// TIA Portal V17 export
// export: Created 2026-04-13T11:12:41.6152652Z, ExportSetting WithDefaults, DisplayName Totally Integrated Automation Portal, DisplayVersion V17 Update 4, DisplayName TIA Portal Openness, DisplayVersion V17 Update 4, DisplayName TIA Portal Version Control Interface, DisplayVersion V17, DisplayName SINAMICS Startdrive Advanced, DisplayVersion V17, DisplayName SINAMICS Startdrive G130, G150, S120, S150, SINAMICS MV, S210, DisplayVersion V17, DisplayName SINAMICS Startdrive G110M, G120, G120C, G120D, G120P, G115D, DisplayVersion V17, DisplayName STEP 7 Professional, DisplayVersion V17 Update 4, DisplayName STEP 7 Safety, DisplayVersion V17, DisplayName WinCC Professional, DisplayVersion V17 Update 4
FUNCTION_BLOCK "A4-蠕动泵控制"   // FB9, SCL
{ S7_Optimized_Access := 'TRUE' }
VERSION : 0.1
// stored: AutoNumber true, IsIECCheckEnabled false, IsRetainMemResEnabled false, MemoryReserve 100, SetENOAutomatically false, UDAEnableTagReadback false
   VAR_INPUT
      HMI上限 : Real := 50.0;
      HMI下限 : Real;
      PLC上限 : Int := 27648;
      PLC下限 : Int := 0;
      泵报警信号 : Bool;
      泵输入电流 : Int;
   END_VAR
   VAR_OUTPUT
      泵输出反馈 : Real;
      泵报警输出 : Bool;
   END_VAR
   VAR_IN_OUT
      模式设定 : Real;
      泵控制按钮 : Bool;
      频率设定 : Real;
      泵输出Q : Bool;
      泵速度AO : Int;
      安全停机 : Bool;
      泵正反转按钮 : Bool;
      泵正反输出 : Bool;
      动画 : Int;
   END_VAR
   VAR
      Temp_1 : Int;
      DBD1 : Real;
      DBD2 : Real;
      DBD3 : Real;
   END_VAR
BEGIN

   //手动控制--------------------------------------------------------------------------------------------------------------
   IF #模式设定 = 2.0 OR #模式设定 = 3.0 OR #模式设定 = 4.0 THEN
       //预热器加热手动控制
       IF #泵控制按钮 THEN
           #泵输出Q := TRUE;
           (* #泵速度AO := REAL_TO_INT((#频率设定 - #工程下限) * (#模拟高限 - #模拟低限) / (#工程上限 - #工程下限) + #模拟低限); *)
           (* #泵速度AO := REAL_TO_INT(#频率设定 * 27648.0 / 50.0); *)
           #DBD1 := NORM_X_REAL(MIN := #HMI下限, VALUE := #频率设定, MAX := #HMI上限);
           #泵速度AO := SCALE_X_INT(MIN := #PLC下限, VALUE := #DBD1, MAX := #PLC上限);
       ELSE
           #泵输出Q := FALSE;
       END_IF;

       IF #泵正反转按钮 THEN
           #泵正反输出 := 1;
       ELSE
           #泵正反输出 := 0;
       END_IF;
   END_IF;

   //自动启动--------------------------------------------------------------------------------------------------------------


   IF #模式设定 = 1.0 THEN
       (* #泵速度AO := REAL_TO_INT((#频率设定 - #工程下限) * (#模拟高限 - #模拟低限) / (#工程上限 - #工程下限) + #模拟低限); *)
       (* #泵速度AO := REAL_TO_INT(#频率设定 * 27648.0 / 50.0); *)
       #DBD2 := NORM_X_REAL(MIN := #HMI下限, VALUE := #频率设定, MAX := #HMI上限);
       #泵速度AO := SCALE_X_INT(MIN := #PLC下限, VALUE := #DBD2, MAX := #PLC上限);



   END_IF;


   IF #泵输出Q THEN
       #DBD3 := NORM_X_REAL(MIN := #PLC下限, VALUE := #泵输入电流, MAX := #PLC上限);
       #泵输出反馈 := SCALE_X_REAL(MIN := #HMI下限, VALUE := #DBD3, MAX := #HMI上限);
   ELSE
       #泵输出反馈 := 0;
   END_IF;

   IF #泵报警信号 THEN
       #泵报警输出 := TRUE;
   ELSE
       #泵报警输出 := FALSE;
   END_IF;


   IF #泵报警信号 THEN
       #泵报警输出 := TRUE;
   ELSE
       #泵报警输出 := FALSE;
   END_IF;

   IF #泵报警输出 THEN
       #泵速度AO := 0;
       #泵控制按钮 := FALSE;
       #泵输出Q := FALSE;
   END_IF;
   IF #模式设定 = 1 AND #泵报警输出 THEN

       #安全停机 := 1;
   END_IF;


   IF #泵输出Q AND #频率设定 > 1 THEN
       IF "Clock_10Hz" THEN
           #Temp_1 := #Temp_1 + 1;
       END_IF;

       IF #Temp_1 =2 THEN
           #Temp_1 := 0;
       END_IF;
       IF #Temp_1 = 0 THEN
           #动画 := 0;
       END_IF;
       IF #Temp_1 = 1 THEN

           #动画 := 1;
       END_IF;

   END_IF;
   IF NOT #泵输出Q THEN
       #动画 := 0;
   END_IF;
END_FUNCTION_BLOCK
